FUNCTION_BLOCK FB_LEDS (* An orientable array of rectangular LEDs *)
  (* Standard: 61499-1 *)
  (* Version 0.0, 2003-11-22, JHC, Rockwell Automation, Derived from FB_BAR. *)
  (* Compiler header: package fb.rt.hmi; import java.awt.*; *)
  (* Compiler Java IBM VisualAge 3.0 *)
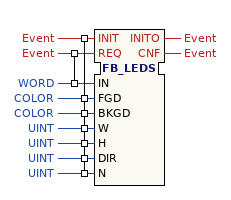
  EVENT_INPUT
    INIT WITH FGD, BKGD, W, H, DIR, N; (* Initialization Request *)
    REQ WITH IN; (* Update the bar *)
  END_EVENT
  EVENT_OUTPUT
    INITO; (* Initialization Confirm *)
    CNF; (* REQ Confirmation *)
  END_EVENT
  VAR_INPUT
    IN : WORD; (* Bits to display(up to 16) *)
    FGD : COLOR := yellow; (* Foreground Color *)
    BKGD : COLOR := black; (* Background Color *)
    W : UINT := 100; (* Bar width *)
    H : UINT := 25; (* Bar height *)
    DIR : UINT; (* Orientation:0=L/R,1=T/B,2=R/L,3=B/T *)
    N : UINT := 1; (* Number of bits to display,starting with LSB-Internally limited to 0<N<17 *)
  END_VAR
END_FUNCTION_BLOCK
